ADAPTER ASRT (* unidirectional Adapter Interface for 3 Events *)
  (* Standard: 61499-1; Description: Copyright (c) 2026 HR Agrartechnik GmbH This program and the accompanying materials are made available under the terms of the Eclipse Public License 2.0 which is available at https://www.eclipse.org/legal/epl-2.0/ SPDX-License-Identifier: EPL-2.0 *)
  (* Version 1.0, 2026-09-03, Franz Höpfinger, HR Agrartechnik GmbH, Initial Version, wie ASR (2 Events) aber mit TOGGLE, fuer AX_T_FF_SR *)
  PACKAGE adapter::types::unidirectional;
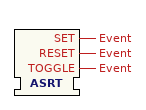
  EVENT_OUTPUT
    SET; (* Set / Switch on *)
    RESET; (* Reset / Switch off *)
    TOGGLE; (* Toggle / Switch output *)
  END_EVENT
END_ADAPTER
